SUBAPPLICATION F_PWM_RAW_TO_PERCENT (* Fieldbus-Rohwert (DINT, 0-64255) in PWM-Sollwert-Anteil (REAL 0.0-1.0) umrechnen, Gegenstueck zu F_PWM_PERCENT_TO_RAW, fuer RampLimitFS.OUT *)
  (* Standard: 61499-2 *)
  (* Version 1.0, 2026-08-28, franz *)
  PACKAGE MyLib::sys;
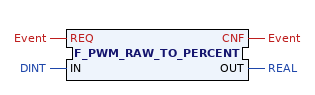
  EVENT_INPUT
    REQ; (* Normal Execution Request *)
  END_EVENT
  EVENT_OUTPUT
    CNF; (* Execution Confirmation *)
  END_EVENT
  VAR_INPUT
    IN : DINT; (* Fieldbus-Rohwert 0-64255 (0x0000-0xFAFF, SAE J1939/ISO 11783 VALID_SIGNAL_W), z.B. RampLimitFS.OUT *)
  END_VAR
  VAR_OUTPUT
    OUT : REAL; (* Sollwert-Anteil 0.0-1.0 (nicht Prozent 0-100!), mit 100.0 multiplizieren fuer Prozent-Anzeige *)
  END_VAR
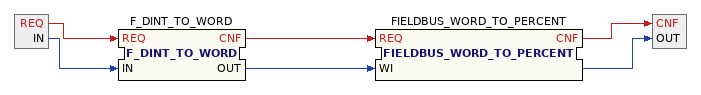
  FBS
    F_DINT_TO_WORD : iec61131::conversion::F_DINT_TO_WORD;
    FIELDBUS_WORD_TO_PERCENT : eclipse4diac::signalprocessing::FIELDBUS_WORD_TO_PERCENT;
  END_FBS
  EVENT_CONNECTIONS
    REQ TO F_DINT_TO_WORD.REQ;
    F_DINT_TO_WORD.CNF TO FIELDBUS_WORD_TO_PERCENT.REQ;
    FIELDBUS_WORD_TO_PERCENT.CNF TO CNF;
  END_CONNECTIONS
  DATA_CONNECTIONS
    IN TO F_DINT_TO_WORD.IN;
    F_DINT_TO_WORD.OUT TO FIELDBUS_WORD_TO_PERCENT.WI;
    FIELDBUS_WORD_TO_PERCENT. TO OUT;
  END_CONNECTIONS
END_SUBAPPLICATION
